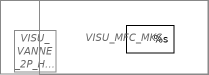
VISUALIZATION VISU_LIGNE_GAZ_VGAUCHE  // 209x75
VAR_IN_OUT
	m_Input_MACHINE:	BLOCK_MODE_MARCHE_V2_0;
	m_Input_MASSFLOW:	BLOCK_MFC_MKS_NoCoE;
	m_Input_LIGNE_GAZ:	BLOCK_LIGNE_GAZ;
END_VAR
    Frame (14,30 42x42)
        shows VISU_VANNE_2P_H_ACT2(m_Input_VANNE := m_Input_LIGNE_GAZ.VGI)
    Rectangle (126,25 48x28), "%s", text variable: m_Input_MASSFLOW.CONF_Util_Name
    Frame (39,0 170x75)
        shows VISU_MFC_MKS(m_Input_MACHINE := m_Input_MACHINE, m_Input_MASSFLOW := m_Input_MASSFLOW, m_Input_LIGNE_GAZ := m_Input_LIGNE_GAZ)
        p3089095539: m_Input_MACHINE
        p1532468285: m_Input_MASSFLOW
        p4266626122: m_Input_LIGNE_GAZ
END_VISUALIZATION

(* stored: Version 1.1.0.1, ProductVersion 3.1.4024.12
   Visu VISU_LIGNE_GAZ_VGAUCHE: Id {2050368c-1e14-43c3-8628-234ac15a5b17} *)
